/// Dummy IO for virtual axis.
TYPE ST_AxisVirtualIO :
STRUCT
	stIn: ST_AxisIn;
	stOut: ST_AxisOut;
END_STRUCT
END_TYPE

(* stored: Version 1.1.0.1, ProductVersion 3.1.4020.12
   DUT ST_AxisVirtualIO: Id {28fcb924-cc9f-47d4-92b7-c057a3f0aea8} *)
